(*
SPDX-FileCopyrightText: © 2026 Oleksandr Tiutyk <trofimich@gmail.com>
SPDX-License-Identifier: MIT
License: https://opensource.org/license/mit
*)

(*!
<summary>Receives this library namespace from the TwinCAT compiler.</summary>
<description>
The init_namespace attribute initializes CurrentNamespace before ordinary library calls. This passive
internal helper performs no cyclic work and owns no dynamic resources. Its namespace output is read-only
by contract and remains valid while the containing instance is alive.
</description>
*)

{attribute 'no_explicit_call' := 'do not call this function block directly'}
FUNCTION_BLOCK INTERNAL NamespaceExtractor
VAR_OUTPUT
	//! <summary>Compiler-initialized namespace; callers borrow this storage without modifying it.</summary>
	{attribute 'init_namespace'} 
	CurrentNamespace : STRING; 	
END_VAR

END_FUNCTION_BLOCK

(* stored: Version 1.1.0.1
   POU NamespaceExtractor: Id {24cd2545-f1b6-4072-926d-c02c3a970344}, SpecialFunc None *)
